# B&R Automation Studio project TestProjectDay1
Automation Studio 4.12.8.41 SP; technology packages: mappCockpit 5.24.4, mappMotion 5.29.0, mappView 5.24.4

## Configuration MainCPU

CPU X20CP3687X, AutomationRuntime O4.93, Build 4.1.2, Safety 0.0, Vc 

### Task classes (Cpu.sw)
```
Cyclic#4:
  Conveyor <- MachineControl.Conveyor.prg
  PiperLogic <- MachineControl.PiperLogic.prg
  Pusher <- MachineControl.Pusher.prg
DataObjects: McAcpSys
NcDataObjects: McDriveLog
Binaries: arsvcreg, udbdef, McAcpDrv, arflatprv, McProfGen, arcoal, FWRules, TCData, McAcpSim, ashwd, Config_1, ashwac, User, sysconf, asfw, arconfig, iomap, Role
Libraries: operator, astime, AsIecCon, standard, sys_lib, brsystem, runtime, McBase, MpBase, McAcpAx, McAxis, MpAxis, csvfilelib, fiowrap, hmitools, logthat, piper, ringbuflib, stringext, FileIO, AsBrStr, AsArLog, AsBrWStr, ArEventLog, powerlnk, asepl, CoTrace, AsZip
```

### Hardware
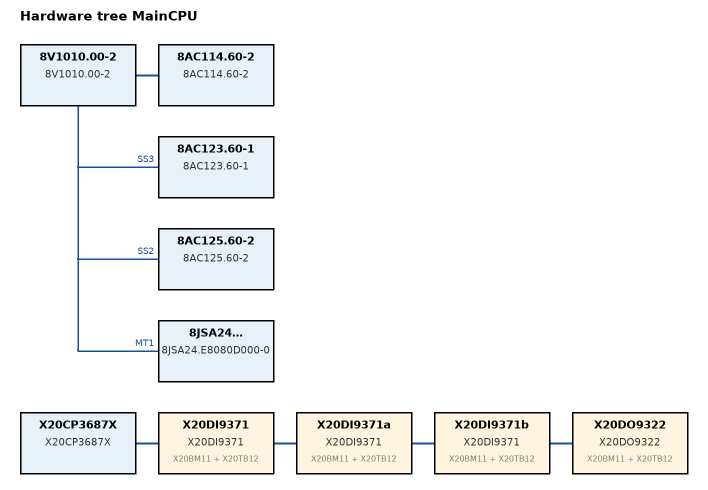
```
8AC114.60-2 : 8AC114.60-2 v1.0.0.8  [SS -> 8V1010.00-2.SS1; PLK1 -> X20CP3687X.IF3 (NodeNumber=1) [Cable Type=PowerlinkCable, Length=10, Version=1.0.0.3]]
8AC123.60-1 : 8AC123.60-1 v2.2.0.0  [SS -> 8V1010.00-2.SS3]
  PlugInType = Encoder
  McAcoposTypeID = AcoposPlugInConfig
  LinesPerRevolution = 0
  IgnoreCheck = 0
8AC125.60-2 : 8AC125.60-2 v2.2.0.0  [SS -> 8V1010.00-2.SS2]
  PlugInType = Encoder
  McAcoposTypeID = AcoposPlugInConfig
  NumberOfLeadingZeros = 0
  NumberOfPositionBits = 17
  NumberOfTrailingZeros = 0
  StatusBit1 = 6
  StatusBit2 = 6
  CRCpolynomial = 67
  IncrementsPerRevolution = 131072
8JSA24.E8080D000-0 : 8JSA24.E8080D000-0 v1.0.6.30  [MT -> 8V1010.00-2.MT1]
8V1010.00-2 : 8V1010.00-2 v2.2.0.0
  DriveConfiguration/Module:
    McAcoposTypeID = AcoposConfig
    ActivateACOPOSSimulationOnPLC = 0
  DriveConfiguration/Channel[1]/RealAxis:
    AxisReference = gAxis_1
    MechanicalElementsIsInvisible = 0
  DriveConfiguration/Channel[1]/RealAxis/MechanicalElements/Gearbox:
    InputIsReadOnly = 0
    Input = 1
    OutputIsReadOnly = 0
    Output = 1
  DriveConfiguration/Channel[1]/RealAxis/MechanicalElements/RotaryToLinearTransformation:
    ReferenceDistanceIsReadOnly = 0
    ReferenceDistance = 1
  DriveConfiguration/Channel[1]/RealAxis/Controller:
    ModeIsReadOnly = 0
    Mode = PositionController
  DriveConfiguration/Channel[1]/RealAxis/Controller/Mode/Position:
    ProportionalGain = 50.0
    IntegrationTime = 0.0
    PredictionTime = 0.0004
    TotalDelayTime = 0.0004
  DriveConfiguration/Channel[1]/RealAxis/Controller/Mode/Speed:
    ProportionalGainIsReadOnly = 0
    ProportionalGain = 2.0
    IntegrationTimeIsReadOnly = 0
    IntegrationTime = 0.0
    FilterTimeIsReadOnly = 0
    FilterTime = 0.0
  DriveConfiguration/Channel[1]/RealAxis/Controller/Mode/LoopFilters:
    LoopFilterXIsReadOnly = 0
    LoopFilter1 = NotUsed
    LoopFilter2 = NotUsed
    LoopFilter3 = NotUsed
  DriveConfiguration/Channel[1]/RealAxis/Homing:
    ModeIsReadOnly = 0
    Mode = Direct
  DriveConfiguration/Channel[1]/RealAxis/Homing/Mode:
    Position = 0.0
    ReferencePulse = NotUsed
  DriveConfiguration/Channel[1]/RealAxis/Homing:
    RestorePositionVariable = 
  DriveConfiguration/Channel[1]/RealAxis/StopReaction:
    QuickstopIsReadOnly = 0
    Quickstop = DecelerationLimit
    DriveErrorIsReadOnly = 0
    DriveError = DecelerationLimit
    FilterTime = 0.0
  DriveConfiguration/Channel[1]/RealAxis/MovementErrorLimits:
    PositionError = 1.0
    VelocityErrorMonitoring = Automatic1
  DriveConfiguration/Channel[1]/RealAxis:
    JerkFilterIsReadOnly = 0
    JerkFilter = NotUsed
    ZeroVibrationFilter = NotUsed
  DriveConfiguration/Channel[1]/RealAxis/DigitalInputs/HomingSwitch:
    SourceIsReadOnly = 0
    Source = X1Ref
    Level = High
  DriveConfiguration/Channel[1]/RealAxis/DigitalInputs/PositiveLimitSwitch:
    Source = X1PosLim
    Level = High
  DriveConfiguration/Channel[1]/RealAxis/DigitalInputs/NegativeLimitSwitch:
    Source = X1NegLim
    Level = High
  DriveConfiguration/Channel[1]/RealAxis/DigitalInputs/Trigger1:
    Source = X1Trigger1
    Level = High
  DriveConfiguration/Channel[1]/RealAxis/DigitalInputs/Trigger2:
    Source = X1Trigger2
    Level = High
  DriveConfiguration/Channel[1]/RealAxis/DigitalInputs/Quickstop:
    Input = Trigger2
  DriveConfiguration/Channel[1]/RealAxis/Simulation:
    SimulationModeOnPLC = SetValueGeneration
    SimulationModeOnACOPOS = NotUsed
  DriveConfiguration/Channel[1]:
    ExternalEncoderAxis = NotUsed
X20BM11 : X20BM11 v1.1.0.0  [X2X1 -> X20CP3687X.IF6]
X20BM11a : X20BM11 v1.1.0.0  [X2X1 -> X20BM11.X2X2]
X20BM11b : X20BM11 v1.1.0.0  [X2X1 -> X20BM11a.X2X2]
X20BM11c : X20BM11 v1.1.0.0  [X2X1 -> X20BM11b.X2X2]
X20CP3687X : X20CP3687X v1.6.2.0
  Connector IF2:
    ActivateDevice = 1
    ActivateSnmp = 2
  ConfigurationID = TestProjectDay1_MainCPU
  FileDevice1
  FileDeviceName1 = USER
  FileDevicePath1 = USER_PATH
  ActivateOpcUa = 1
  OpcUa_AuthenticationSecurityPolicy_EnableNone = 1
  OpcUa_AuthenticationSecurityPolicy_EnableBasic128Rsa15 = 1
  OpcUaInformationModels_PV_Version = 1
X20DI9371 : X20DI9371 v1.6.0.0  [SS1 -> X20TB12.SS; SL -> X20BM11.SL1]
X20DI9371a : X20DI9371 v1.6.0.0  [SS1 -> X20TB12a.SS; SL -> X20BM11a.SL1]
X20DI9371b : X20DI9371 v1.6.0.0  [SS1 -> X20TB12b.SS; SL -> X20BM11b.SL1]
X20DO9322 : X20DO9322 v1.7.0.0  [SS1 -> X20TB12c.SS; SL -> X20BM11c.SL1]
X20TB12 : X20TB12 v1.0.0.0
X20TB12a : X20TB12 v1.0.0.0
X20TB12b : X20TB12 v1.0.0.0
X20TB12c : X20TB12 v1.0.0.0
```

### Config_1.axis - X20CP3687X/mappMotion/Config_1.axis
```
Element gAxis_1 (Type=axis)
  BaseTypeIsReadOnly = 0
  BaseType = LinearBounded
    MeasurementUnit = 5066068
    MeasurementResolutionIsReadOnly = 0
    MeasurementResolution = 0.01
    CountDirectionIsReadOnly = 0
    CountDirection = Standard
  MovementLimitsIsReadOnly = 0
  MovementLimits = Internal
    Position:
      LowerLimitMin = -1.79769313486231E308
      UpperLimitMax = 1.79769313486231E308
      LowerLimit = 0
      UpperLimit = 500
    VelocityIsReadOnly = 0
    Velocity:
      VelocityMax = 3.4E38
      Velocity = 10.0
    AccelerationIsReadOnly = 0
    Acceleration:
      AccelerationMax = 3.4E38
      Acceleration = 50.0
    DecelerationIsReadOnly = 0
    Deceleration:
      DecelerationMax = 3.4E38
      Deceleration = 50.0
  Alarms = None
```

## Logical view

Binary libraries used (declarations not repeated): operator, runtime, astime, AsIecCon, standard, sys_lib, brsystem, McBase 5.29.0, MpBase, McAcpAx 5.29.0, McAxis 5.29.0, MpAxis 5.29.0, csvfilelib, fiowrap, hmitools, logthat, piper, ringbuflib, stringext, FileIO, AsBrStr, AsArLog, AsBrWStr, ArEventLog, CoTrace, AsZip

### Global.var - Global variables
```iecst
VAR
	mode : USINT;
	gMachine : Piper_typ;
END_VAR
```

### IO.typ
```iecst
TYPE
	IO_Pusher_typ : 	STRUCT
		aoActualPosition : REAL;
		diPusherExtended : BOOL;
		extendedTimer : TON;
		state : PusherState;
		reset : BOOL;
		diPusherRetracted : BOOL;
	END_STRUCT;
	IO_typ : 	STRUCT
		conveyor : ARRAY[0..MAI_CONVEYORS]OF IO_Conveyor_typ;
		spawnCase : BOOL;
		pusher : IO_Pusher_typ;
	END_STRUCT;
	StateEnum :
		(
		ST_BOOTING,
		ST_SINGOUT,
		ST_SINGIN,
		ST_IDLE,
		ST_HOLD
		);
	PusherState :
		(
		ST_BOOT,
		ST_INIT,
		ST_WAIT,
		ST_PUSH,
		ST_PULL
		);
	IO_Conveyor_typ : 	STRUCT
		diPhotoeyeEntrance : BOOL;
		diPhotoeyeExit : BOOL;
		doRunForward : BOOL;
		doRunReverse : BOOL;
		_diPhotoeye2 : BOOL;
		_diPhotoeye1 : BOOL;
		singoutTimer : TON;
		singinTimer : TON;
		state : StateEnum;
		diPhotoeye2 : BOOL;
		diPhotoeye1 : BOOL;
		downstreamReadyToReceive : BOOL;
		upstreamReadyToSend : BOOL;
		readyToReceive : BOOL;
		readyToSend : BOOL;
		runMotor : BOOL;
		singinHoldTimer : TON;
		aoRunSpeed : REAL;
	END_STRUCT;
END_TYPE
```

### IO.var
```iecst
VAR
	io : IO_typ;
END_VAR
VAR CONSTANT
	MAX_CONVEYORS : UDINT := 4;
	MAI_CONVEYORS : UDINT := MAX_CONVEYORS-1;
END_VAR
VAR
	i : UDINT;
END_VAR
```


### Program Logical/MachineControl/Conveyor (IEC)

#### Types.typ
```iecst
TYPE
	stateENUM2 :
		(
		ST_RUNNING,
		ST_DONE,
		ST_STOP
		);
END_TYPE
```

#### Variables.var
```iecst
VAR
	counter : INT;
	spawnTimer : TON;
	direction : BOOL;
	CounterDone : BOOL;
	startCounting : BOOL;
	state : stateENUM2;
	machineStart : BOOL;
	machineStop : BOOL;
	machineRunning : BOOL;
END_VAR
```

#### Cyclic.st
```iecst
PROGRAM _CYCLIC
	(* Insert code here *)

//	IF diPhotoeye = FALSE THEN
//		doPusher := TRUE;
//	END_IF
	PiperInterface;

	CASE state OF

		ST_STOP:
			counter := 0;
			IF startCounting THEN
				state := ST_RUNNING;
			END_IF
		ST_RUNNING:
			counter := counter +1;
			IF counter> 500 THEN
				CounterDone := TRUE;
				state := ST_DONE;
			END_IF
		ST_DONE:
		 // Do nothing

	END_CASE

	// Set mode for operation
	mode := 4;

	IF machineStart THEN
		io.conveyor[0].state := ST_IDLE;
		io.conveyor[1].state := ST_IDLE;
		io.conveyor[2].state := ST_IDLE;
		io.conveyor[3].state := ST_IDLE;
	ELSIF machineStop THEN
		io.conveyor[0].state := ST_BOOTING;
		io.conveyor[1].state := ST_BOOTING;
		io.conveyor[2].state := ST_BOOTING;
		io.conveyor[3].state := ST_BOOTING;
	END_IF

	IF machineRunning AND (spawnTimer.Q AND NOT io.conveyor[0].diPhotoeyeEntrance) AND NOT (io.conveyor[0].state = ST_SINGIN) THEN
		io.spawnCase := TRUE;
		spawnTimer.IN := FALSE;
	ELSE
		io.spawnCase := FALSE;
		spawnTimer.IN := TRUE;
	END_IF

	FOR i := 0 TO MAI_CONVEYORS DO

		// Zone timers
		io.conveyor[i].singinTimer();
		io.conveyor[i].singoutTimer();
		io.conveyor[i].singinTimer.PT := T#6s;
		io.conveyor[i].singoutTimer.PT := T#1200ms;

		IF mode = 2 THEN
			IF io.conveyor[0].diPhotoeyeEntrance THEN
				direction := TRUE;
			END_IF
			IF io.conveyor[3].diPhotoeyeExit THEN
				direction := FALSE;
			END_IF
		END_IF

		// defining signals
		IF mode = 2 THEN
			IF NOT direction THEN
				io.conveyor[i].diPhotoeye1 := io.conveyor[i].diPhotoeyeExit;
				io.conveyor[i].diPhotoeye2 := io.conveyor[i].diPhotoeyeEntrance;
				io.conveyor[i].doRunReverse := io.conveyor[i].runMotor;
				io.conveyor[i].doRunForward := FALSE;
			ELSE
				io.conveyor[i].diPhotoeye1 := io.conveyor[i].diPhotoeyeEntrance;
				io.conveyor[i].diPhotoeye2 := io.conveyor[i].diPhotoeyeExit;
				io.conveyor[i].doRunForward := io.conveyor[i].runMotor;
				io.conveyor[i].doRunReverse := FALSE;
			END_IF
		ELSE
			io.conveyor[i].diPhotoeye1 := io.conveyor[i].diPhotoeyeEntrance;
			io.conveyor[i].diPhotoeye2 := io.conveyor[i].diPhotoeyeExit;
			io.conveyor[i].doRunForward := io.conveyor[i].runMotor;
			io.conveyor[i].doRunReverse := FALSE;
		END_IF

		// Ready to send signal definition for different modes
		IF mode = 2 THEN
			IF io.conveyor[i].diPhotoeye2 AND io.conveyor[i].singinHoldTimer.Q THEN
				io.conveyor[i].readyToSend := TRUE;
			ELSE
				io.conveyor[i].readyToSend := FALSE;
			END_IF
		ELSE
			IF io.conveyor[i].diPhotoeye2 THEN
				io.conveyor[i].readyToSend := TRUE;
			ELSE
				io.conveyor[i].readyToSend := FALSE;
			END_IF
		END_IF

		// Ready to Receieve signal definition for different modes
		IF NOT io.conveyor[i].diPhotoeye2 AND io.conveyor[i].state = ST_IDLE THEN
			io.conveyor[i].readyToReceive := TRUE;
		ELSE
			io.conveyor[i].readyToReceive := FALSE;
		END_IF

		//handshakes for both directions

		IF i = 0 THEN
			io.conveyor[i].upstreamReadyToSend := io.conveyor[i].diPhotoeye1;
		ELSE
			io.conveyor[i].upstreamReadyToSend := io.conveyor[i-1].readyToSend;
		END_IF

		IF i = MAI_CONVEYORS THEN
			IF mode = 2 THEN
				io.conveyor[i].downstreamReadyToReceive := FALSE;
			ELSE
				io.conveyor[i].downstreamReadyToReceive := TRUE;
			END_IF
		ELSE
			io.conveyor[i].downstreamReadyToReceive := io.conveyor[i+1].readyToReceive;
		END_IF

		CASE io.conveyor[i].state OF
			ST_BOOTING:
				// DO NOTHING
				io.conveyor[i].runMotor := FALSE;
				io.conveyor[i].singoutTimer.IN := FALSE;
				io.conveyor[i].singinTimer.IN := FALSE;

			ST_IDLE:
				io.conveyor[i].runMotor := FALSE;
				io.conveyor[i].singoutTimer.IN := FALSE;
				io.conveyor[i].singinTimer.IN := FALSE;

				IF  io.conveyor[i].upstreamReadyToSend AND io.conveyor[i].readyToReceive THEN
					io.conveyor[i].state := ST_SINGIN;
				END_IF

			ST_SINGIN :
						io.conveyor[i].runMotor := TRUE ;
						io.conveyor[i].singinTimer.IN := TRUE;

						IF io.conveyor[i].diPhotoeye2 THEN
							io.conveyor[i].singinTimer.IN := FALSE;
							io.conveyor[i].runMotor := FALSE;
							io.conveyor[i].singinHoldTimer.IN := TRUE;

							IF io.conveyor[i].downstreamReadyToReceive THEN
								IF mode = 3 AND io.conveyor[i].singinHoldTimer.Q THEN
									io.conveyor[i].state := ST_SINGOUT;
								ELSE
									io.conveyor[i].state := ST_HOLD;
								END_IF
							ELSE
								io.conveyor[i].state := ST_HOLD;
				            END_IF
				END_IF

						IF 	io.conveyor[i].singinTimer.Q THEN
							io.conveyor[i].state := ST_IDLE;
							io.conveyor[i].singinTimer.IN := FALSE;
						END_IF

			ST_SINGOUT:

						io.conveyor[i].runMotor := TRUE;
						io.conveyor[i].singoutTimer.IN := TRUE;
						io.conveyor[i].singinHoldTimer.IN := FALSE;

						IF NOT io.conveyor[i].diPhotoeye2 THEN
							io.conveyor[i].singinTimer.IN := FALSE;
							io.conveyor[i].runMotor := FALSE;
							io.conveyor[i].state := ST_IDLE;
						END_IF

			ST_HOLD:

						io.conveyor[i].runMotor := FALSE;
						io.conveyor[i].singoutTimer.IN := FALSE;
						io.conveyor[i].singinTimer.IN := FALSE;
                        io.conveyor[i].singinHoldTimer.IN := FALSE;

						IF io.conveyor[i].downstreamReadyToReceive THEN
							io.conveyor[i].state := ST_SINGOUT;
						END_IF

		END_CASE
		//One shot logic
		io.conveyor[i]._diPhotoeye1 := io.conveyor[i].diPhotoeye1;
		io.conveyor[i]._diPhotoeye2 := io.conveyor[i].diPhotoeye2;

	END_FOR

	// Multiple timers and axis function calls

	spawnTimer(PT:= T#8s);

END_PROGRAM
```

#### Init.st
```iecst
PROGRAM _INIT
	(* Insert code here *)
	counter := 0;
	io.pusher.state := ST_INIT;
	state := ST_STOP;

END_PROGRAM
```

#### PiperInterface.st
```iecst
ACTION PiperInterface:

	//Give this module a name so it is easier to debug
	ModuleInterface.ModuleName:=	'Conveyor';

	//Add a module to the Piper
	Module.ModuleInterface:=	ADR(ModuleInterface);
	Module.Piper:= 	ADR(gMachine);
	Module();

	// Handle any machine states that this module needs to respond to
	CASE ModuleInterface.PiperState OF
		//		MACH_ST_BOOTING:
		  //MACH_ST_CLEARING:

		MACH_ST_STOPPED:
			machineStop := FALSE;

		MACH_ST_STARTING:
			machineStart := TRUE;
			ModuleInterface.ModuleResponse:=	ModuleInterface.PiperState;
		//MACH_ST_IDLE:
		//		MACH_ST_SUSPENDED:
		MACH_ST_EXECUTE:
			machineStart := FALSE;
			machineRunning := TRUE;

		MACH_ST_STOPPING:
			machineStop := TRUE;
			machineRunning := FALSE;
			ModuleInterface.ModuleResponse:=	ModuleInterface.PiperState;
		//		MACH_ST_ABORTING:
		//MACH_ST_ABORTED:
			//		MACH_ST_HOLDING:
		//		MACH_ST_HELD:
		//		MACH_ST_UNHOLDING:
		//		MACH_ST_SUSPENDING:
		//		MACH_ST_UNSUSPENDING:
		//MACH_ST_RESETTING:

		//		MACH_ST_COMPLETING:
		//		MACH_ST_COMPLETE:

		MACH_ST_BYPASSED:

		ELSE
			ModuleInterface.ModuleResponse:=	ModuleInterface.PiperState;

	END_CASE
END_ACTION
```

### Program Logical/MachineControl/Pusher (IEC)

#### Cyclic.st - Cyclic code
```iecst
PROGRAM _CYCLIC
	(* Insert code here *)
	io.pusher.aoActualPosition := 100*LREAL_TO_REAL(axisHandler.Position);
	axisHandler.MpLink := ADR(gAxis_1);
	axisHandler.Parameters :=  ADR(axisParameters);
	axisHandler.Enable := TRUE;

	// commands from PIPER to cyclic
	IF machineStop THEN
		axisHandler.Home:= TRUE;
		io.pusher.state := ST_BOOT;
	END_IF

	PiperInterface;

	// If mode 4 is selected run pusher logic
	IF mode = 4 THEN
		CASE io.pusher.state OF
			ST_BOOT:
				// Do nothing

				IF machineStart THEN
					io.pusher.state := ST_INIT;
				END_IF
			ST_INIT:
				machineStart := FALSE;

				IF axisHandler.Active AND NOT axisHandler.PowerOn THEN
					axisHandler.Power := TRUE;
				ELSIF axisHandler.PowerOn AND NOT axisHandler.Home THEN
					axisHandler.Home:= TRUE;
				ELSIF axisHandler.IsHomed THEN
					io.pusher.state := ST_WAIT;
				END_IF

			ST_WAIT:
				axisHandler.Home:= FALSE;
				IF io.conveyor[2].diPhotoeye1 AND io.conveyor[2].doRunForward THEN
					boxLengthTimer.IN := TRUE;
					IF boxLengthTimer.ET > T#600ms THEN
						io.pusher.state := ST_PUSH;
					END_IF
				ELSE
					boxLengthTimer.IN := FALSE;
				END_IF

			ST_PUSH :
				axisParameters.Position := 5.0;
				axisParameters.Velocity := 5.0;
				axisParameters.Acceleration := 25.0;
				axisParameters.Deceleration := 25.0;
				axisHandler.MoveAbsolute := TRUE;
				io.pusher.extendedTimer.IN := TRUE;
				boxLengthTimer.IN := FALSE;

				IF axisHandler.Position = axisParameters.Position OR io.pusher.extendedTimer.Q THEN
					axisHandler.MoveAbsolute := FALSE;
					io.pusher.extendedTimer.IN := FALSE;
					io.pusher.state := ST_PULL;
				END_IF

			ST_PULL:

				axisHandler.Home:= TRUE;
				IF axisHandler.IsHomed THEN
					axisHandler.Home:= TRUE;
					io.pusher.state := ST_WAIT;
				END_IF
		END_CASE
	END_IF

	axisHandler();
	io.pusher.extendedTimer(PT := T#3s);
	boxLengthTimer(PT := T#1S);
END_PROGRAM
```

#### Init.st - Init code
```iecst
PROGRAM _INIT
	(* Insert code here *)
	 io.pusher.state := ST_BOOT;
END_PROGRAM
```

#### Variables.var - Local variables
```iecst
VAR
	axisParameters : MpAxisBasicParType;
	axisHandler : MpAxisBasic;
	boxLengthTimer : TON;
	machineStart : BOOL;
	machineStop : BOOL;
END_VAR
```

#### PiperInterface.st
```iecst
ACTION PiperInterface:

	//Give this module a name so it is easier to debug
	ModuleInterface.ModuleName:=	'Pusher';

	//Add a module to the Piper
	Module.ModuleInterface:=	ADR(ModuleInterface);
	Module.Piper:= 	ADR(gMachine);
	Module();

	// Handle any machine states that this module needs to respond to
	CASE ModuleInterface.PiperState OF
		//		MACH_ST_BOOTING:
		//      MACH_ST_CLEARING:
		MACH_ST_STOPPED:
			machineStop := FALSE;
			ModuleInterface.ModuleResponse:=	ModuleInterface.PiperState;
		MACH_ST_STARTING:
			machineStart := TRUE;
			IF axisHandler.IsHomed THEN
				ModuleInterface.ModuleResponse:=	ModuleInterface.PiperState;
			END_IF

			// MACH_ST_IDLE:
			//		MACH_ST_SUSPENDED:
		MACH_ST_EXECUTE:
			machineStart := FALSE;

		MACH_ST_STOPPING:
			machineStop := TRUE;
			IF axisHandler.IsHomed THEN
				ModuleInterface.ModuleResponse:=	ModuleInterface.PiperState;
			END_IF
		//		MACH_ST_ABORTING:
		//      MACH_ST_ABORTED:

		//		MACH_ST_HOLDING:
		//		MACH_ST_HELD:
		//		MACH_ST_UNHOLDING:
		//		MACH_ST_SUSPENDING:
		//		MACH_ST_UNSUSPENDING:
		MACH_ST_RESETTING:
			io.pusher.reset := TRUE;
			ModuleInterface.ModuleResponse:=	ModuleInterface.PiperState;
			//		MACH_ST_COMPLETING:
		//		MACH_ST_COMPLETE:

		MACH_ST_BYPASSED:

		ELSE
			ModuleInterface.ModuleResponse:=	ModuleInterface.PiperState;

	END_CASE
END_ACTION
```

#### PiperModuleTemplate.var
```iecst
VAR
	ModuleInterface : Module_Interface_typ;
	Module : Piper_Module_Fub;
END_VAR

VAR CONSTANT

END_VAR
```

### Program Logical/MachineControl/PiperLogic (IEC)

#### Cyclic.st - Cyclic code
```iecst
PROGRAM _CYCLIC
	(* Insert code here *)
	Piper_fn_Cyclic(gMachine);

END_PROGRAM
```

#### Init.st - Init code
```iecst
PROGRAM _INIT
	(* Insert code here *)

END_PROGRAM
```

#### Variables.var - Local variables
```iecst
VAR
	startCounting : BOOL;
	state : stateENUM2;
	counter : DINT;
END_VAR
```

#### PiperInterface.st
```iecst
ACTION PiperInterface:

	//Give this module a name so it is easier to debug
	ModuleInterface.ModuleName:=	'Counter';

	//Add a module to the Piper
	Module.ModuleInterface:=	ADR(ModuleInterface);
	Module.Piper:= 	ADR(gMachine);
	Module();

	// Handle any machine states that this module needs to respond to
	CASE ModuleInterface.PiperState OF
		//		MACH_ST_BOOTING:
		MACH_ST_CLEARING:
			startCounting := TRUE;
			ModuleInterface.ModuleResponse:=	ModuleInterface.PiperState;
		//		MACH_ST_STOPPED:
		//		MACH_ST_STARTING:
		//		MACH_ST_IDLE:
		//		MACH_ST_SUSPENDED:
		//	    MACH_ST_EXECUTE:
		//		MACH_ST_STOPPING:
		//		MACH_ST_ABORTING:
		//		MACH_ST_ABORTED:
		//		MACH_ST_HOLDING:
		//		MACH_ST_HELD:
		//		MACH_ST_UNHOLDING:
		//		MACH_ST_SUSPENDING:
		//		MACH_ST_UNSUSPENDING:
		//		MACH_ST_RESETTING:
		//		MACH_ST_COMPLETING:
		//		MACH_ST_COMPLETE:

		MACH_ST_BYPASSED:

		ELSE
			ModuleInterface.ModuleResponse:=	ModuleInterface.PiperState;

	END_CASE
END_ACTION
```

### Program Logical/MachineControl/Program

#### Types.typ
```iecst
TYPE
	CountEnum :
		(
		ST_RUNNING,
		ST_WAIT
		);
	edge_Detection_Typ : 	STRUCT
		_diPhotoeyeExit : BOOL;
		_diPhotoeyeEntrance : BOOL;
		Occupied : BOOL;
		Timer : TON;
		singoutTimer : TON;
		singinTimer : TON;
		readyToSend : BOOL;
		upstreamReadyToSend : BOOL;
		downstreamReadyToReceive : BOOL;
		DirectionForward : BOOL;
		readyToReceive : BOOL;
	END_STRUCT;
END_TYPE
```

#### Variables.var
```iecst
VAR
	counterState : CountEnum;
	counter : INT;
	diPhotoeye : BOOL;
	doPusher : BOOL;
	myCommand : BOOL;
	convPhotoeyePrev : ARRAY[0..MAI_CONVEYORS] OF edge_Detection_Typ;
	testTimer : TON;
	test : INT;
	spawnTimer : TON;
	direction : BOOL;
	mode : INT;
END_VAR
```

#### Cyclic.st
```iecst
PROGRAM _CYCLIC
	(* Insert code here *)

//	IF diPhotoeye = FALSE THEN
//		doPusher := TRUE;
//	END_IF

//	testTimer();

//  Below peice of logic was added to test case statement testing during day 1.
//
//	CASE counterState OF
//		ST_WAIT:
//		     IF testTimer.Q THEN
//					counterState := ST_RUNNING;
//			END_IF
//
//	    ST_RUNNING:
//			    counter := counter + 1;
//				testTimer.IN := FALSE;
//			    counterState := ST_WAIT;
//	END_CASE
//    //test :=  counter MOD 10;
	//myCommand := (test = 0) AND (counter<200)

// Start of Conveyor logic

	io.conveyor[i].singinTimer.PT := T#6s;

	CASE mode OF
		1:

	    // Regular mode - Day 1

			IF spawnTimer.Q AND NOT io.conveyor[0].diPhotoeyeEntrance THEN
				io.spawnCase := TRUE;
				spawnTimer.IN := FALSE;
			ELSE
				io.spawnCase := FALSE;
				spawnTimer.IN := TRUE;
			END_IF
			// Handshakes

			FOR i := 0 TO MAI_CONVEYORS DO

				// defining signals
				    io.conveyor[i].diPhotoeye1 := io.conveyor[i].diPhotoeyeEntrance;
					io.conveyor[i].diPhotoeye2 := io.conveyor[i].diPhotoeyeExit;
					io.conveyor[i].doRunForward := io.conveyor[i].runMotor;
					io.conveyor[i].doRunReverse := FALSE;

				IF io.conveyor[i].diPhotoeye2 THEN
					io.conveyor[i].readyToSend := TRUE;
				ELSE
					io.conveyor[i].readyToSend := FALSE;
				END_IF

				IF NOT io.conveyor[i].diPhotoeye2 THEN
					io.conveyor[i].readyToReceive := TRUE;
				ELSE
					io.conveyor[i].readyToReceive := FALSE;
				END_IF

					IF i = 0 THEN
						io.conveyor[i].upstreamReadyToSend := io.conveyor[i].diPhotoeye1;
					ELSE
						io.conveyor[i].upstreamReadyToSend := io.conveyor[i-1].readyToSend;
					END_IF

					IF i = MAI_CONVEYORS THEN
						io.conveyor[i].downstreamReadyToReceive := FALSE;
					ELSE
						io.conveyor[i].downstreamReadyToReceive := io.conveyor[i+1].readyToReceive;
					END_IF

				CASE io.conveyor[i].state OF
					ST_IDLE:
						io.conveyor[i].runMotor := FALSE;
						io.conveyor[i].singoutTimer.IN := FALSE;
						io.conveyor[i].singinTimer.IN := FALSE;

						IF  io.conveyor[i].upstreamReadyToSend AND io.conveyor[i].readyToReceive THEN
							io.conveyor[i].state := ST_SINGIN;
						END_IF

					ST_SINGIN :
						io.conveyor[i].runMotor := TRUE ;
						io.conveyor[i].singinTimer.IN := TRUE;

						IF io.conveyor[i].diPhotoeye2 THEN
							io.conveyor[i].runMotor := FALSE;
							IF io.conveyor[i].downstreamReadyToReceive THEN
								io.conveyor[i].state := ST_SINGOUT;
							ELSE
								io.conveyor[i].state := ST_HOLD;
							END_IF
						END_IF

					ST_SINGOUT:

						io.conveyor[i].runMotor := TRUE;
						io.conveyor[i].singoutTimer.IN := TRUE;

						IF NOT io.conveyor[i].diPhotoeye2 THEN
							io.conveyor[i].singinTimer.IN := FALSE;
							io.conveyor[i].runMotor := FALSE;
							io.conveyor[i].state := ST_IDLE;
						END_IF

					ST_HOLD:

						io.conveyor[i].runMotor := FALSE;
						io.conveyor[i].singoutTimer.IN := FALSE;
						io.conveyor[i].singinTimer.IN := FALSE;

						IF io.conveyor[i].downstreamReadyToReceive THEN
							io.conveyor[i].state := ST_SINGOUT;
						END_IF

				END_CASE

				io.conveyor[i]._diPhotoeye1 := io.conveyor[i].diPhotoeye1;
				io.conveyor[i]._diPhotoeye2 := io.conveyor[i].diPhotoeye2;

			END_FOR
		2:

			// toggle between forward reverse

			// Logic to change box direction when it hits last zone on each side

			IF io.conveyor[0].diPhotoeyeEntrance THEN
				direction := TRUE;
			END_IF

			IF io.conveyor[3].diPhotoeyeExit THEN
				direction := FALSE;
	     	END_IF
			// Handshakes

			FOR i := 0 TO MAI_CONVEYORS DO

				IF direction THEN
					io.conveyor[i].diPhotoeye1 := io.conveyor[i].diPhotoeyeEntrance;
					io.conveyor[i].diPhotoeye2 := io.conveyor[i].diPhotoeyeExit;
					io.conveyor[i].doRunForward := io.conveyor[i].runMotor;
					io.conveyor[i].doRunReverse := FALSE;
				ELSE
					io.conveyor[i].diPhotoeye1 := io.conveyor[i].diPhotoeyeExit;
					io.conveyor[i].diPhotoeye2 := io.conveyor[i].diPhotoeyeEntrance;
					io.conveyor[i].doRunReverse := io.conveyor[i].runMotor;
					io.conveyor[i].doRunForward := FALSE;
				END_IF

				IF io.conveyor[i].diPhotoeye2 THEN
					io.conveyor[i].readyToSend := TRUE;
				ELSE
					io.conveyor[i].readyToSend := FALSE;
				END_IF

				IF NOT io.conveyor[i].diPhotoeye2 THEN
					io.conveyor[i].readyToReceive := TRUE;
				ELSE
					io.conveyor[i].readyToReceive := FALSE;
				END_IF

				IF direction THEN
						IF i = 0 THEN
					    	io.conveyor[i].upstreamReadyToSend := io.conveyor[i].diPhotoeye1;
						ELSE
							io.conveyor[i].upstreamReadyToSend := io.conveyor[i-1].readyToSend;
						END_IF

						IF i = MAI_CONVEYORS THEN
							io.conveyor[i].downstreamReadyToReceive := FALSE;
						ELSE
							io.conveyor[i].downstreamReadyToReceive := io.conveyor[i+1].readyToReceive;
						END_IF
				ELSE
					IF i = MAI_CONVEYORS THEN
						io.conveyor[i].upstreamReadyToSend := io.conveyor[i].diPhotoeye2;
					ELSE
						io.conveyor[i].upstreamReadyToSend := io.conveyor[i+1].readyToSend;
					END_IF

					IF i = 0 THEN
						io.conveyor[i].downstreamReadyToReceive := FALSE;
					ELSE
						io.conveyor[i].downstreamReadyToReceive := io.conveyor[i-1].readyToReceive;
					END_IF
				END_IF

				CASE io.conveyor[i].state OF
					ST_IDLE:
						io.conveyor[i].runMotor := FALSE;
					    io.conveyor[i].singoutTimer.IN := FALSE;
						io.conveyor[i].singinTimer.IN := FALSE;

						IF  io.conveyor[i].upstreamReadyToSend AND io.conveyor[i].readyToReceive THEN
							io.conveyor[i].state := ST_SINGIN;
						END_IF

					ST_SINGIN :
						io.conveyor[i].runMotor := TRUE ;
						io.conveyor[i].singinTimer.IN := TRUE;

						IF io.conveyor[i].diPhotoeye2 THEN
							io.conveyor[i].runMotor := FALSE;
							IF io.conveyor[i].downstreamReadyToReceive THEN
								io.conveyor[i].state := ST_SINGOUT;
							ELSE
								io.conveyor[i].state := ST_HOLD;
							END_IF
						END_IF

					ST_SINGOUT:

						io.conveyor[i].runMotor := TRUE;
						io.conveyor[i].singoutTimer.IN := TRUE;

						IF NOT io.conveyor[i].diPhotoeye2 THEN
							io.conveyor[i].singinTimer.IN := FALSE;
							io.conveyor[i].runMotor := FALSE;
							io.conveyor[i].state := ST_IDLE;
						END_IF

					ST_HOLD:

						io.conveyor[i].runMotor := FALSE;
						io.conveyor[i].singoutTimer.IN := FALSE;
						io.conveyor[i].singinTimer.IN := FALSE;

						IF io.conveyor[i].downstreamReadyToReceive THEN
							io.conveyor[i].state := ST_SINGOUT;
						END_IF

				END_CASE

				io.conveyor[i]._diPhotoeye1 := io.conveyor[i].diPhotoeye1;
				io.conveyor[i]._diPhotoeye2 := io.conveyor[i].diPhotoeye2;

			END_FOR

		3:

			END_FOR
	END_CASE

END_PROGRAM
```

#### Init.st
```iecst
PROGRAM _INIT
	(* Insert code here *)
	counter := 0;

END_PROGRAM
```

Listed in the project but not available here: Logical/Global.typ, Logical/MachineControl/Pusher/Exit.st, Logical/MachineControl/Pusher/Types.typ, Logical/MachineControl/PiperLogic/Exit.st, Logical/MachineControl/PiperLogic/Types.typ, Logical/MachineControl/PiperLogic/PiperModuleTemplate.var
